TYPE ST_00_StationStructTemplate :
STRUCT

	e00SeqState		: E_00_StationStateTemplate;

	REQ				: ST_STATION_Requests;
	STAT				: ST_STATION_Status;

(*Variable examles only*)
(*
	bPassthroughMode			:BOOL;

	stBundleTracking				: ST_BundleTrackingRegister;
	bTrigCamera					: BOOL;
	bCameraDone					: BOOL;


*)

END_STRUCT
END_TYPE

(* stored: Version 1.1.0.1, ProductVersion 3.1.4024.15
   DUT ST_00_StationStructTemplate: Id {3f2083c8-d543-48dc-9e65-6fbde5a50fa8} *)
